RoboDK station: Kinema_primeros_pasos.rdk

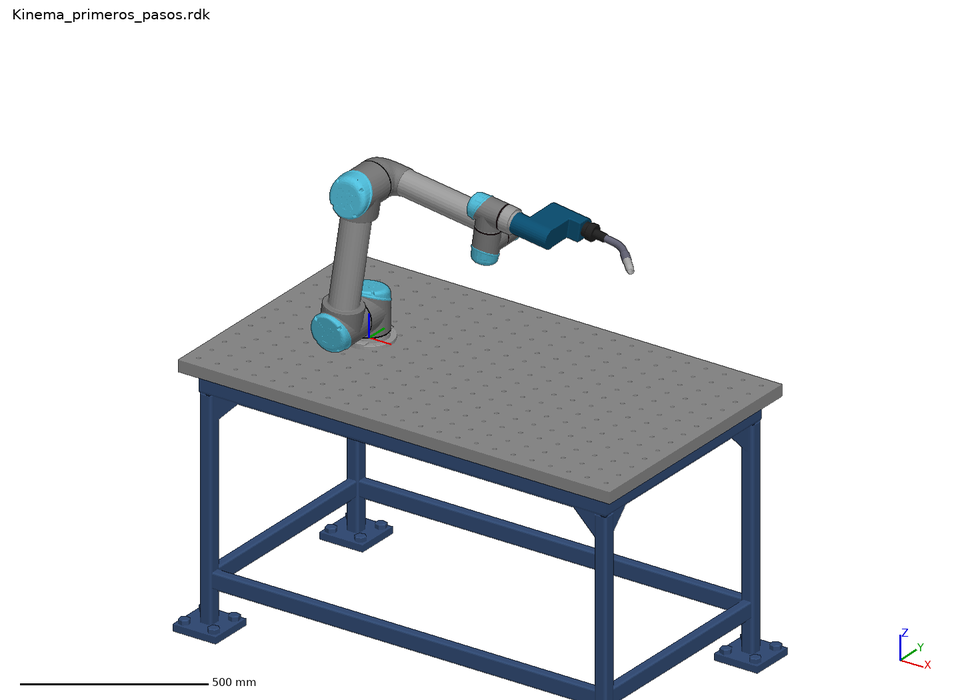
[picture v0: the station drawn from its stored meshes, robots at their saved joint values, targets as dots, program paths as lines]
Station Kinema_primeros_pasos (saved by RoboDK 5.9.4). Poses are relative to the parent item; angles as X-Y-Z fixed-axis rotations.
  - frame UR5 Base at (0, 0, 0) mm
    - robot UR5: 6 axes
        modified DH rows (alpha deg, a mm, theta deg, d mm): 0, 0, 0, 89.2; 90, 0, 180, 0; 0, 425, 0, 0; 0, 392, 0, 109.3; -90, 0, 0, 94.75; 90, 0, 180, 82.5
        joint limits [-360, -360, -360, -360, -360, -360] to [360, 360, 360, 360, 360, 360]; home [0, -90, -90, 0, 90, 0]; saved at [0.938, -98.438, -90, 0, 90, 0]
      - tool Generic Welding Gun (Over-arm), TCP at (-4, 0, 371.3) mm, rotated rx 0 ry 45 rz 0 deg, size 169.7 x 60 x 367 mm
  - object Table 1400x800x800mm at (0, 0, 0) mm, size 1420 x 820 x 800 mm, geometry from Table-1400x800x800mm.sld
  - folder Programas
    - program Iniciar (1 instructions, listed below)
    - Python program Movimiento (listed below)
  - Python program Prog3 (listed below)

--- program Iniciar (robot UR5) ---
  Ejecutar Movimiento

--- Python program Movimiento ---
from robodk import robolink
from robodk import robomath

from robolink import *
from robodk import *

import json
import time

# -----------------------------
# Conexión con RoboDK
# -----------------------------
RDK = Robolink()

robot = RDK.Item('UR5')

if not robot.Valid():
    raise Exception("No se encontró el robot.")

robot.setSpeed(10, 10)

# Guardamos la posición Home
home = robot.Joints()

# Variables para evitar mover continuamente
ultima_x = None
ultima_y = None

while True:

    # Leer JSON
    try:

        with open(r"C:\Users\aaron\Documents\KINEMA_NEXUS\data\robot_data.json", "r") as f:
            datos = json.load(f)

    except (json.JSONDecodeError, FileNotFoundError):
        time.sleep(0.05)
        continue

    x = datos["x"]
    y = datos["y"]

    # Solo mover si cambia la posición
    if ultima_x is None or abs(x-ultima_x) > 2 or abs(y-ultima_y) > 2:

        print(f"X = {x:.1f} mm   Y = {y:.1f} mm")

        # ---------------------------------------------------
        # PRUEBA
        # ---------------------------------------------------
        # De momento convertimos X e Y a pequeños movimientos
        # articulares únicamente para comprobar la comunicación.
        # ---------------------------------------------------

        j1 = x * 0.1
        j2 = -90 + y * 0.05

        robot.MoveJ([j1,j2,-90,0,90, 0])

        ultima_x = x
        ultima_y = y

    time.sleep(0.05)

--- Python program Prog3 ---
from robodk.robolink import *
from robodk.robomath import *

import json

RDK = Robolink()

robot = RDK.Item('UR5')

with open(r"C:\Users\aaron\Documents\KINEMA_NEXUS\data\robot_data.json","r") as f:
    datos = json.load(f)

print(datos)

from robodk.robomath import *

x = datos["x"]
y = datos["y"]

z = 300          # altura fija

pose = transl(x, y, z)

robot.MoveL(pose)
